// Mitsubishi GX Works2 project: Servo   PLC: Q03UD

PROGRAM IOCHECK
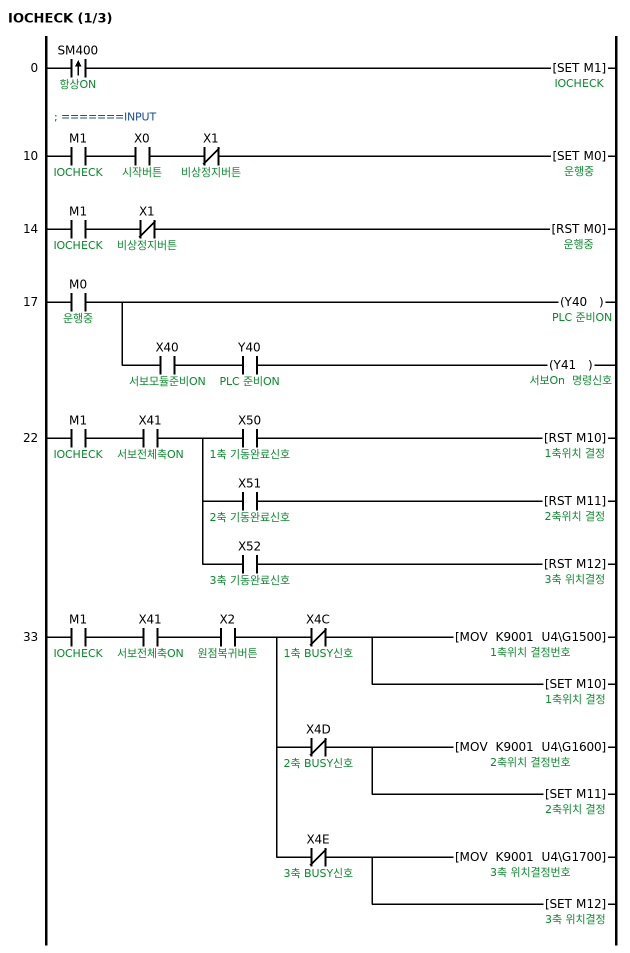
0     LDP     SM400  ; 항상ON
      SET     M1  ; IOCHECK
; =======INPUT
10    LD      M1  ; IOCHECK
      AND     X0  ; 시작버튼
      ANI     X1  ; 비상정지버튼
      SET     M0  ; 운행중
14    LD      M1  ; IOCHECK
      ANI     X1  ; 비상정지버튼
      RST     M0  ; 운행중
17    LD      M0  ; 운행중
      OUT     Y40  ; PLC 준비ON
      AND     X40  ; 서보모듈준비ON
      AND     Y40  ; PLC 준비ON
      OUT     Y41  ; 서보On  명령신호
22    LD      M1  ; IOCHECK
      AND     X41  ; 서보전체축ON
      MPS
      AND     X50  ; 1축 기동완료신호
      RST     M10  ; 1축위치 결정
      MRD
      AND     X51  ; 2축 기동완료신호
      RST     M11  ; 2축위치 결정
      MPP
      AND     X52  ; 3축 기동완료신호
      RST     M12  ; 3축 위치결정
33    LD      M1  ; IOCHECK
      AND     X41  ; 서보전체축ON
      AND     X2  ; 원점복귀버튼
      MPS
      ANI     X4C  ; 1축 BUSY신호
      MOV     K9001 U4\G1500  ; 1축위치 결정번호
      SET     M10  ; 1축위치 결정
      MRD
      ANI     X4D  ; 2축 BUSY신호
      MOV     K9001 U4\G1600  ; 2축위치 결정번호
      SET     M11  ; 2축위치 결정
      MPP
      ANI     X4E  ; 3축 BUSY신호
      MOV     K9001 U4\G1700  ; 3축 위치결정번호
      SET     M12  ; 3축 위치결정
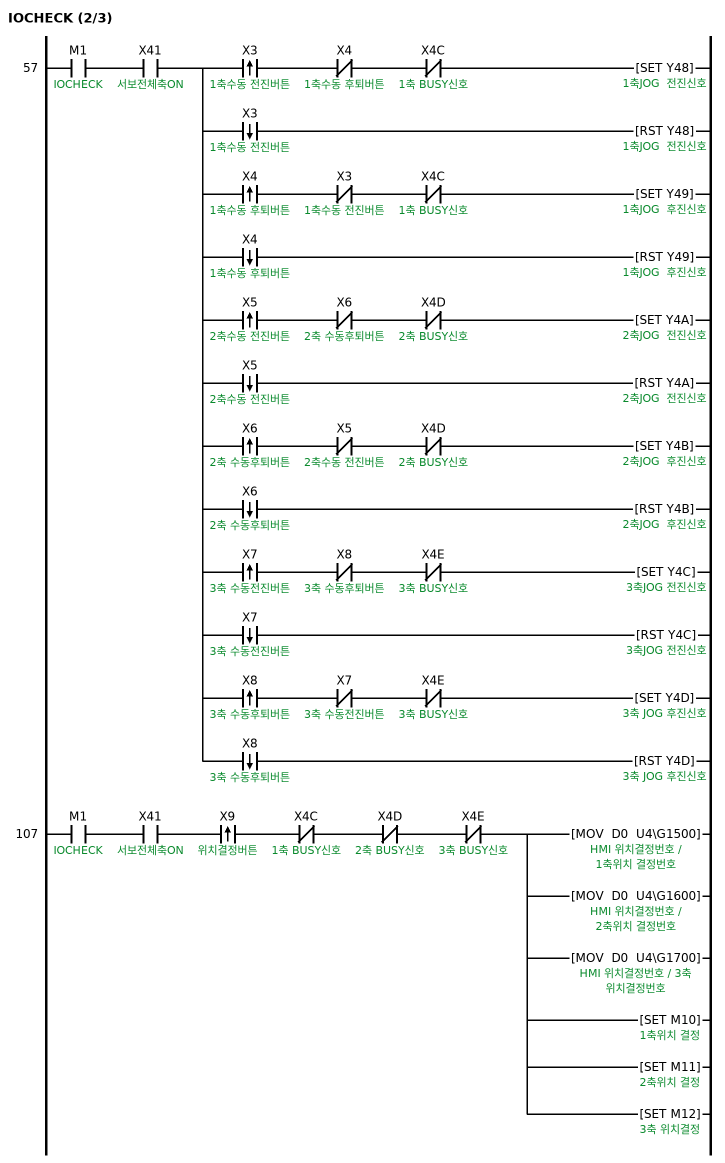
57    LD      M1  ; IOCHECK
      AND     X41  ; 서보전체축ON
      MPS
      ANDP    X3  ; 1축수동 전진버튼
      ANI     X4  ; 1축수동 후퇴버튼
      ANI     X4C  ; 1축 BUSY신호
      SET     Y48  ; 1축JOG  전진신호
      MRD
      ANDF    X3  ; 1축수동 전진버튼
      RST     Y48  ; 1축JOG  전진신호
      MRD
      ANDP    X4  ; 1축수동 후퇴버튼
      ANI     X3  ; 1축수동 전진버튼
      ANI     X4C  ; 1축 BUSY신호
      SET     Y49  ; 1축JOG  후진신호
      MRD
      ANDF    X4  ; 1축수동 후퇴버튼
      RST     Y49  ; 1축JOG  후진신호
      MRD
      ANDP    X5  ; 2축수동 전진버튼
      ANI     X6  ; 2축 수동후퇴버튼
      ANI     X4D  ; 2축 BUSY신호
      SET     Y4A  ; 2축JOG  전진신호
      MRD
      ANDF    X5  ; 2축수동 전진버튼
      RST     Y4A  ; 2축JOG  전진신호
      MRD
      ANDP    X6  ; 2축 수동후퇴버튼
      ANI     X5  ; 2축수동 전진버튼
      ANI     X4D  ; 2축 BUSY신호
      SET     Y4B  ; 2축JOG  후진신호
      MRD
      ANDF    X6  ; 2축 수동후퇴버튼
      RST     Y4B  ; 2축JOG  후진신호
      MRD
      ANDP    X7  ; 3축 수동전진버튼
      ANI     X8  ; 3축 수동후퇴버튼
      ANI     X4E  ; 3축 BUSY신호
      SET     Y4C  ; 3축JOG 전진신호
      MRD
      ANDF    X7  ; 3축 수동전진버튼
      RST     Y4C  ; 3축JOG 전진신호
      MRD
      ANDP    X8  ; 3축 수동후퇴버튼
      ANI     X7  ; 3축 수동전진버튼
      ANI     X4E  ; 3축 BUSY신호
      SET     Y4D  ; 3축 JOG 후진신호
      MPP
      ANDF    X8  ; 3축 수동후퇴버튼
      RST     Y4D  ; 3축 JOG 후진신호
107   LD      M1  ; IOCHECK
      AND     X41  ; 서보전체축ON
      ANDP    X9  ; 위치결정버튼
      ANI     X4C  ; 1축 BUSY신호
      ANI     X4D  ; 2축 BUSY신호
      ANI     X4E  ; 3축 BUSY신호
      MOV     D0 U4\G1500  ; HMI 위치결정번호
      MOV     D0 U4\G1600
      MOV     D0 U4\G1700
      SET     M10  ; 1축위치 결정
      SET     M11  ; 2축위치 결정
      SET     M12  ; 3축 위치결정
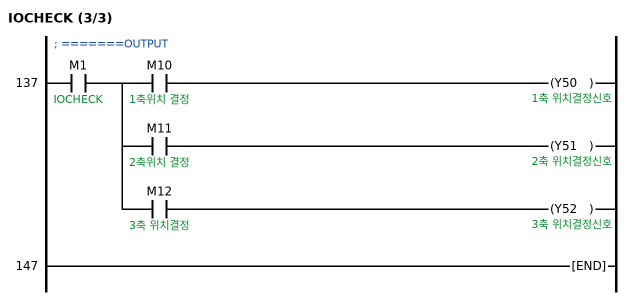
; =======OUTPUT
137   LD      M1  ; IOCHECK
      MPS
      AND     M10  ; 1축위치 결정
      OUT     Y50  ; 1축 위치결정신호
      MRD
      AND     M11  ; 2축위치 결정
      OUT     Y51  ; 2축 위치결정신호
      MPP
      AND     M12  ; 3축 위치결정
      OUT     Y52  ; 3축 위치결정신호
147   END
END_PROGRAM

PROGRAM MAIN
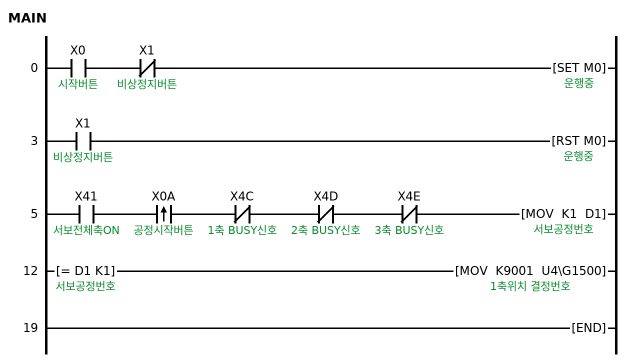
0     LD      X0  ; 시작버튼
      ANI     X1  ; 비상정지버튼
      SET     M0  ; 운행중
3     LD      X1  ; 비상정지버튼
      RST     M0  ; 운행중
5     LD      X41  ; 서보전체축ON
      ANDP    X0A  ; 공정시작버튼
      ANI     X4C  ; 1축 BUSY신호
      ANI     X4D  ; 2축 BUSY신호
      ANI     X4E  ; 3축 BUSY신호
      MOV     K1 D1  ; 서보공정번호
12    LD=     D1 K1  ; 서보공정번호
      MOV     K9001 U4\G1500  ; 1축위치 결정번호
19    END
END_PROGRAM
